INTERFACE I_Base EXTENDS __SYSTEM.IQueryInterface

END_INTERFACE

(* stored: Version 1.1.0.1, ProductVersion 3.1.4026.18
   Itf I_Base: Id {75b7395a-241b-44d7-9e71-5c854c3777a7} *)
